// TIA Portal project "StepperMotor" (V18)

(* hardware
DEVICE "S7-1200 station_1"  S7-1200 Station
   slot 0: "Rack_0"  S7-1200 Rack  Rack  V1.0
   slot 1: "PLC_1"  CPU 1212C DC/DC/DC  6ES7 212-1AE40-0XB0  V4.2
*)

// ===== PLC "PLC_1"  CPU 1212C DC/DC/DC =====

VAR_GLOBAL   // PLC tag table "Default tag table"
   "Axis_1_Pulse" AT %Q0.0 : Bool;
   "Axis_1_Direction" AT %Q0.1 : Bool;
   "EnableStepper" AT %M1.0 : Bool;
   "JogFwd" AT %M10.0 : Bool;
   "JogBck" AT %M10.1 : Bool;
   "Execute" AT %M1.1 : Bool;
   "EStop" AT %I0.0 : Bool;
   "Velocity" AT %MD4 : Real;
   "Switch Up" AT %I0.1 : Bool;
   "Switch Down" AT %I0.2 : Bool;
   "Green PB" AT %I0.3 : Bool;
   "Red PB" AT %I0.4 : Bool;
   "ONS3" AT %M0.0 : Bool;
   "ONS4" AT %M0.1 : Bool;
   "StepperDisable" AT %Q0.2 : Bool;
END_VAR

// folder: System blocks/Program resources

DATA_BLOCK "IEC_Timer_0_DB"   // DB4
{ S7_Optimized_Access := 'TRUE' }
AUTHOR : Simatic
FAMILY : IEC
NAME : IEC_TMR
VERSION : 1.0
// stored: InstanceOfName IEC_TIMER
"IEC_TIMER"
BEGIN
END_DATA_BLOCK

// folder: (top level)

DATA_BLOCK "Axis_1"   // DB1, Motion_DB
{ S7_Optimized_Access := 'TRUE' }
AUTHOR : SIMATIC
FAMILY : BasicMC
NAME : TO_PosAx
VERSION : 6.0
// stored: InstanceOfName TO_PositioningAxis
"TO_PositioningAxis"
BEGIN
   // Axis.DirectionOutputEnabledCU = TRUE
   // Axis.OnlinePtoModeCU = 16#0000_0002
   // Axis.SelectedChannel2EnumCU = %Q0.1
   // Axis.SelectedChannel1EnumCU = %Q0.0
   // Pulse.MinDeltaDeltaFrequencyCU = 0.004
   // Pulse.MaxDeltaDeltaFrequencyCU = 1.0E+10
   // Pulse.MinDeltaFrequencyCU = 0.005
   // Pulse.MaxDeltaFrequencyCU = 9.5E+9
   // Pulse.MinFrequencyCU = 1.0
   // Pulse.MaxFrequencyCU = 100000.0
   // Pulse.OutputSourceCU = 16#0000_0000
   // Axis.SelectPTO = 0
   // Axis.LengthUnit.LastDistance = -1
   // Axis.LengthUnitNormalized.Time = 1
   // Axis.LengthUnitNormalized.Distance = -2
   // Axis.Encoder.SelectedHscIndexCU = -1
END_DATA_BLOCK

ORGANIZATION_BLOCK "Main"   // OB1, LAD, ProgramCycle
TITLE = "Main Program Sweep (Cycle)"
{ S7_Optimized_Access := 'TRUE' }
VERSION : 0.1
   VAR_INPUT
      Initial_Call : Bool;   // Initial call of this OB
      Remanence : Bool;   // =True, if remanent data are available
   END_VAR
   VAR_TEMP
      ONS2 : Bool;
      ONS1 : Bool;
   END_VAR
   VAR_TEMP   // added for the SCL form of the ladder/FBD networks
      _w1 : Bool;
      _w2 : Bool;
   END_VAR
BEGIN

REGION Network 1
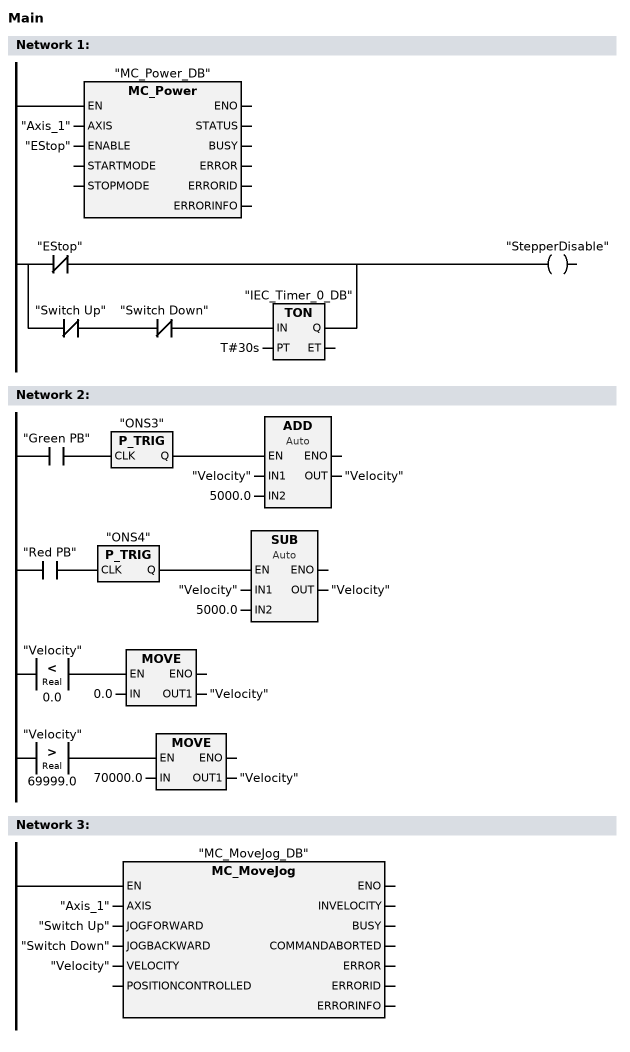
   "MC_Power_DB"(Axis := "Axis_1", Enable := "EStop");   // MC_Power
   "IEC_Timer_0_DB".TON(IN := NOT "Switch Up" AND NOT "Switch Down", PT := T#30s);
   "StepperDisable" := NOT "EStop" OR "IEC_Timer_0_DB".Q;
END_REGION

REGION Network 2
   RUNG wire#powerrail
      Contact( "Green PB" )
      P_Trig( "ONS3" )
      Add(in1 := "Velocity", in2 := 5000.0, out => "Velocity")
   END_RUNG
   RUNG wire#powerrail
      Contact( "Red PB" )
      P_Trig( "ONS4" )
      Sub(in1 := "Velocity", in2 := 5000.0, out => "Velocity")
   END_RUNG
   RUNG wire#powerrail
      { S7_Templates := "SrcType := Real" } LT_Contact(in1 := "Velocity", in2 := 0.0)
      Move(in := 0.0, out1 => "Velocity")
   END_RUNG
   RUNG wire#powerrail
      { S7_Templates := "SrcType := Real" } GT_Contact(in1 := "Velocity", in2 := 69999.0)
      Move(in := 70000.0, out1 => "Velocity")
   END_RUNG
   // the same network as SCL:
   #_w1 := "Green PB" AND NOT "ONS3";   // rising edge
   "ONS3" := "Green PB";
   IF #_w1 THEN "Velocity" := "Velocity" + 5000.0; END_IF;
   #_w2 := "Red PB" AND NOT "ONS4";   // rising edge
   "ONS4" := "Red PB";
   IF #_w2 THEN "Velocity" := "Velocity" - 5000.0; END_IF;
   IF "Velocity" < 0.0 THEN "Velocity" := 0.0; END_IF;
   IF "Velocity" > 69999.0 THEN "Velocity" := 70000.0; END_IF;
END_REGION

REGION Network 3
   "MC_MoveJog_DB"(Axis := "Axis_1",   // MC_MoveJog
                   JogForward := "Switch Up",
                   JogBackward := "Switch Down",
                   Velocity := "Velocity");
END_REGION
END_ORGANIZATION_BLOCK